(* CODESYS project WagoAppKNX.ecp

Project tree, tasks and I/O mapping:
  Steuerung : 750-8202 PFC200 2ETH RS, WAGO, order no. 0750-8202, version 5.11.1.16
    application Application
      libraries: ; WagoAppKNX, * (WAGO)
      task PLC_Task (cyclic, interval t#50ms, priority 15) calls PLC_PRG
      task VISU_TASK (cyclic, interval 100 ms, priority 15) calls VisuElems.Visu_Prg
      program PLC_PRG [CFC]
      visualisation Visualization
    Kbus : Kbus, WAGO, version 1.4.0.2
        unmapped channels: K-BUS diagnostics
      KNX_EIB_TP1_Interface : 075x-16DI, WAGO, order no. 075x-16DI, version 0.0.0.13
          settings: K-BUS Module slot index = 1
          unmapped channels: _IN
      _16_DI_Generic : 075x-16DI, WAGO, order no. 075x-16DI, version 0.0.0.13
          settings: K-BUS Module slot index = 2
          unmapped channels: _IN
      _16_DI_Generic_1 : 075x-16DI, WAGO, order no. 075x-16DI, version 0.0.0.13
          settings: K-BUS Module slot index = 3
          unmapped channels: _IN
      _8_DI_Generic : 075x-8DI, WAGO, order no. 075x-8DI, version 0.0.0.13
          settings: K-BUS Module slot index = 4
          unmapped channels: _IN
      _8_DI_Generic_1 : 075x-8DI, WAGO, order no. 075x-8DI, version 0.0.0.13
          settings: K-BUS Module slot index = 5
          unmapped channels: _IN
      _16_DO_Generic : 075x-16DO, WAGO, order no. 075x-16DO, version 0.0.0.13
          settings: K-BUS Module slot index = 6
          unmapped channels: _OUT
      _16_DO_Generic_1 : 075x-16DO, WAGO, order no. 075x-16DO, version 0.0.0.13
          settings: K-BUS Module slot index = 7
          unmapped channels: _OUT
      _16_DO_Generic_2 : 075x-16DO, WAGO, order no. 075x-16DO, version 0.0.0.13
          settings: K-BUS Module slot index = 8
          unmapped channels: _OUT
      KNX_EIB_TP1_Interface_1 : 0753-0646, WAGO, order no. 0753-0646, version 0.0.0.10
          settings: K-BUS Module slot index = 9
          unmapped channels: _INPUTCHANNEL, _OUTPUTCHANNEL
      DALI_Multi_Master : 0753-0647, WAGO, order no. 0753-0647, version 0.0.0.20
          settings: K-BUS Module slot index = 10
          unmapped channels: _IN, _OUT
    MODBUS
      MODBUS : MODBUS, WAGO, order no. n/a, version 1.1.1.15
    Serial
      COM1 : COM1, WAGO, version 0.0.0.19
  PFC200_2ETH_RS : 750-8202 PFC200 2ETH RS, WAGO, order no. 0750-8202, version 5.14.3.31
    application Application
      libraries: 
      task PLC_Task (cyclic, interval t#50ms, priority 15) calls PLC_PRG
      program PLC_PRG [CFC]
    Kbus : Kbus, WAGO, version 1.4.0.2
        unmapped channels: K-BUS diagnostics
      _8_DI_Generic : 075x-8DI, WAGO, order no. 075x-8DI, version 0.0.0.13
          unmapped channels: _IN
      _2_DO_Generic : 075x-2DO, WAGO, order no. 075x-2DO, version 0.0.0.13
          unmapped channels: _OUT
      KNX_EIB_TP1_Interface : 0753-0646, WAGO, order no. 0753-0646, version 0.0.0.10
          unmapped channels: _INPUTCHANNEL, _OUTPUTCHANNEL
    MODBUS
      MODBUS : MODBUS, WAGO, order no. n/a, version 1.1.1.15
    Serial
      COM1 : COM1, WAGO, version 0.0.0.19
*)

// Steuerung/Application/PLC_PRG
PROGRAM PLC_PRG
VAR
	fbKNX_Master: FbKNX_Master;
	fbKNX_Master_TM: FbKNX_Master_TM;
	oStatus: WagoAppKNX.WagoSysErrorBase.FbResult;
	sStatus: STRING;
	xProgMode: BOOL;
	wCountFbDPT: WORD;
	fbDPT_Switch_Control: WagoAppKNX.FbDPT_Switch_Control;
	xUpdate_PLC: BOOL;
	xControl_OUT: BOOL;
	xSwitch_OUT: BOOL;
	dwIndex_DPT: DWORD;
	xSwitch_IN: BOOL;
	xControl_IN: BOOL;
	xUpdate_KNX: BOOL;
	oStatus_TM: WagoAppKNX.WagoSysErrorBase.FbResult;
	sStatus_TM: STRING;
	stPhyAddress_TM: STRING(9);
	xFilter_Mode_TM: BOOL;
END_VAR

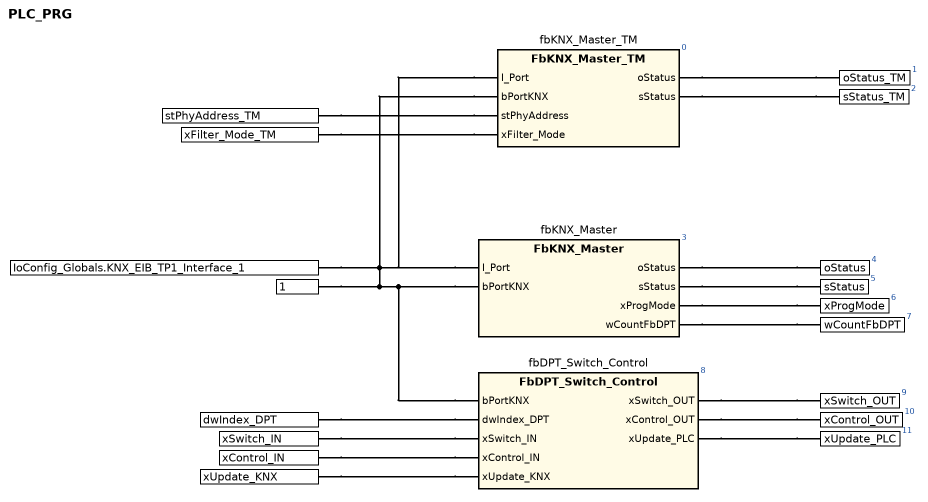
fbKNX_Master_TM(
    I_Port := IoConfig_Globals.KNX_EIB_TP1_Interface_1,
    bPortKNX := 1,
    stPhyAddress := stPhyAddress_TM,
    xFilter_Mode := xFilter_Mode_TM);
oStatus_TM := fbKNX_Master_TM.oStatus;
sStatus_TM := fbKNX_Master_TM.sStatus;
fbKNX_Master(I_Port := IoConfig_Globals.KNX_EIB_TP1_Interface_1, bPortKNX := 1);
oStatus := fbKNX_Master.oStatus;
sStatus := fbKNX_Master.sStatus;
xProgMode := fbKNX_Master.xProgMode;
wCountFbDPT := fbKNX_Master.wCountFbDPT;
fbDPT_Switch_Control(
    bPortKNX := 1,
    dwIndex_DPT := dwIndex_DPT,
    xSwitch_IN := xSwitch_IN,
    xControl_IN := xControl_IN,
    xUpdate_KNX := xUpdate_KNX);
xSwitch_OUT := fbDPT_Switch_Control.xSwitch_OUT;
xControl_OUT := fbDPT_Switch_Control.xControl_OUT;
xUpdate_PLC := fbDPT_Switch_Control.xUpdate_PLC;

END_PROGRAM

// PFC200_2ETH_RS/Application/PLC_PRG
PROGRAM PLC_PRG
VAR
END_VAR

END_PROGRAM

// Steuerung/Application/Visualization
VISUALIZATION Visualization  // 2x2
END_VISUALIZATION
